// TwinCAT 3 PLC project plc
// Title: ExercicesForPlcProgramming
// Company: Beckhoff Automation Belgium
// ProjectVersion: 1.0.0.0
// Description: Exercices of the book Collection of Exercises for PLC Programming by Tom Mejer Antonson ISBN: 978-87-4305-780-2
// ProgramVersion: 3.1.4026.19
// CompilerDefines: VISU_USEPROPERTYINFO
// libraries:
//   Tc2_ControllerToolbox, * (Beckhoff Automation GmbH)
//   Tc2_Standard, * (Beckhoff Automation GmbH)
//   Tc2_System, * (Beckhoff Automation GmbH)
//   VisuDialogs, * (System)
// project tree:
//   Exercises/02. Logical Circuits/ LogicalCircuits.TcPOU, LogicalCircuits_Ex01.TcPOU, LogicalCircuits_Ex02.TcPOU, LogicalCircuits_Ex03.TcPOU, LogicalCircuits_Ex04.TcPOU, LogicalCircuits_Ex05.TcPOU, LogicalCircuits_Ex06.TcPOU, LogicalCircuits_Ex07.TcPOU, LogicalCircuits_Ex08.TcPOU, LogicalCircuits_Ex09.TcPOU, LogicalCircuits_Ex10.TcPOU, LogicalCircuits_Ex11.TcPOU, LogicalCircuits_Ex12.TcPOU
//   Exercises/03. Safety/ Safety.TcPOU, safety_ex01.TcPOU, safety_ex02.TcPOU
//   Exercises/04. Logic and Counters/ logcacounters_ex2.TcPOU, logcacounters_ex3.TcPOU, logcacounters_ex4.TcPOU, logcacounters_ex5.TcPOU, logcacounters_ex6.TcPOU, logcacounters_ex7.TcPOU, LogicAndCounters.TcPOU, LogicandCountersex01.TcPOU
//   Exercises/05. Timers/ Timers.TcPOU, timers_ex01.TcPOU, timers_ex02.TcPOU, timers_ex03.TcPOU, timers_ex04.TcPOU, timers_ex05.TcPOU, timers_ex06.TcPOU
//   Exercises/06. Analog Signals/ AnalogSignals.TcPOU, analogSignals_ex01.TcPOU, analogSignals_ex02.TcPOU, analogSignals_ex03.TcPOU, analogSignals_ex04.TcPOU, analogSignals_ex05.TcPOU, analogSignals_ex06.TcPOU, analogSignals_ex07.TcPOU, FB_Scale.TcPOU, gemiddelde.TcPOU
//   Exercises/07. Applied Mathematics/ AppliedMathematics.TcPOU, appliedmathematics_ex01.TcPOU
//   Exercises/08. Arrays/ Arrays.TcPOU
//   Exercises/09. Functions and Function Blocks/ FunctionsAndFunctionBlocks.TcPOU, FunctionsAndFunctionBlocksex01.TcPOU, FunctionsAndFunctionBlocksex02.TcPOU, FunctionsAndFunctionBlocksex03.TcPOU
//   Exercises/10. Strings and Structs/ StringsAndStructs.TcPOU
//   Exercises/11. Complex Exercises/ ComplexExercises.TcPOU
//   / GlobalTextList.TcGTLO, MAIN.TcPOU, PlcTask.TcTTO, Visualization Manager.TcVMO (not stored)
//   Project Information/ F_GetCompany.TcPOU, F_GetTitle.TcPOU, F_GetVersion.TcPOU
//   Version/ Global_Version.TcGVL
//   _Library/Inputs/GVLs/ GVL_IO.TcGVL
//   _Library/Inputs/POUs/ DigitalInput_NC.TcPOU, MMotor.TcPOU (not stored), motoroef2_12.TcPOU (not stored), Switch_2P.TcPOU, DigitalInput_NO.TcPOU, DigitalOutput.TcPOU, Switch_4P.TcPOU
//   _Library/Inputs/VISUs/ Visualization.TcVIS
//   _Library/ _TemplateFB.TcPOU
// real-time tasks:
//   TASK PlcTask: cycle T#10ms, priority 20, ADS port 350

CONFIGURATION plc
    RESOURCE PLC ON TwinCAT3
        TASK PlcTask(INTERVAL := T#10ms, PRIORITY := 20);
        PROGRAM MAIN WITH PlcTask : MAIN;
    END_RESOURCE
END_CONFIGURATION

// ---- Version/Global_Version.TcGVL
{attribute 'TcGenerated'}
{attribute 'no-analysis'}
{attribute 'linkalways'}
// This function has been automatically generated from the project information.
VAR_GLOBAL CONSTANT
	{attribute 'const_non_replaced'}
	stLibVersion_ExercicesForPlcProgramming : ST_LibVersion := (iMajor := 1, iMinor := 0, iBuild := 0, iRevision := 0, nFlags := 0, sVersion := '1.0.0.0');
END_VAR

// ---- _Library/Inputs/GVLs/GVL_IO.TcGVL
{attribute 'qualified_only'}
VAR_GLOBAL
	// S1						AT %I*: BOOL;		// S14.2
	// S1						: DigitalInput_NO;   	// S14.2
END_VAR

// ---- MAIN.TcPOU
(*
	Simple solutions for the exercices of the book 
	Collection of Exercises for PLC Programming
	by Tom Mejer Antonson
	ISBN: 978-87-4305-780-2
*)
PROGRAM MAIN
VAR
END_VAR

//LogicalCircuits();
//Safety();
//LogicAndCounters();
//Timers();
AnalogSignals();
//AppliedMathematics();
//Arrays();
//FunctionsAndFunctionBlocks();
//StringsAndStructs();
//ComplexExercises();

END_PROGRAM

// ---- Exercises/06. Analog Signals/AnalogSignals.TcPOU
PROGRAM AnalogSignals

analogSignals_ex07();

END_PROGRAM

// ---- Exercises/06. Analog Signals/analogSignals_ex07.TcPOU
PROGRAM analogSignals_ex07
VAR

	weight				: REAL;
	weightsensor		: REAL;
	hoeveelvaliezen		: INT;
	gemiddeldgewicht	: REAL;
	
	OK					: digitalInput_NO;
	Reset				: digitalInput_NO;
	
	tellersmall			: CTU;
	tellernormal		: CTU;
	tellerbig			: CTU;
	telleroversized		: CTU;
	LIN_TRAFO 			: FB_Scale;
	gemiddelde4			: gemiddelde;
	flankok				: R_trig;
END_VAR

flankok(CLK:= ok.isOn, Q=> );

LIN_TRAFO(
	fIN:= weightsensor, 
	fIN_min:= 4, 
	fIN_max:= 20, 
	fOUT_min:= 0, 
	fOUT_max:= 50, 
	fOUT=> weight);
	
//tellers
	tellersmall(
	CU:= (weight > 0.0) AND (weight <= 5) AND (OK.isOn), 
	RESET:= reset.isOn, 
	PV:= , 
	Q=> , 
	CV=> );
	tellernormal(
	CU:= (weight > 5) AND (weight <= 10) AND (OK.isOn), 
	RESET:= reset.isOn, 
	PV:= , 
	Q=> , 
	CV=> );
	tellerbig(
	CU:= (weight > 10) AND (weight <= 20) AND (OK.isOn), 
	RESET:= reset.isOn, 
	PV:= , 
	Q=> , 
	CV=> );
	telleroversized(
	CU:= (weight > 20) AND (weight <=50) AND (OK.isOn), 
	RESET:= reset.isOn, 
	PV:= , 
	Q=> , 
	CV=> );
	
gemiddelde4(
	fValue:= weight, 
	bAdd:= flankok.Q, 
	bReset:= reset.isOn, 
	fAverage=> gemiddeldgewicht, 
	nCount=> hoeveelvaliezen);

END_PROGRAM

// ---- _Library/Inputs/POUs/DigitalInput_NO.TcPOU
{attribute 'no_explicit_call' := 'do not call this POU directly'} 
FUNCTION_BLOCK DigitalInput_NO
VAR
	DI_Input						AT %I*: BOOL;
END_VAR

PROPERTY isOff : bool
GET
isOff 		:= NOT DI_Input;
END_GET
END_PROPERTY

PROPERTY isOn : bool
GET
isOn			:= DI_Input;
END_GET
END_PROPERTY

END_FUNCTION_BLOCK

// ---- Exercises/06. Analog Signals/FB_Scale.TcPOU
FUNCTION_BLOCK FB_Scale
VAR_INPUT
	fIN				: REAL;
	fIN_min 		: REAL;
	fIN_max			: REAL;
	fOUT_min		: REAL;
	fOUT_max 		: REAL;
END_VAR
VAR_OUTPUT
	fOUT 			: REAL;	
END_VAR
VAR
END_VAR

fOUT := fOUT_min + (fIN - fIN_MIN) * (fOUT_max - fOUT_min) / (fIN_max - fIN_min);

END_FUNCTION_BLOCK

// ---- Exercises/06. Analog Signals/gemiddelde.TcPOU
FUNCTION_BLOCK gemiddelde
VAR_INPUT
	fValue : REAL;                     // Waarde om toe te voegen
    bAdd : BOOL;                       // Trigger om waarde toe te voegen
    bReset : BOOL;                     // Reset de berekening
END_VAR
VAR_OUTPUT
	fAverage : REAL;                   // Gemiddelde waarde
    nCount : INT;                      // Aantal metingen
END_VAR
VAR
	 fSum : REAL := 0.0;                // Som van alle waarden
    bAddOld : BOOL := FALSE;           // Voor edge detectie
	
END_VAR

IF bReset THEN
    nCount := 0;
    fSum := 0.0;
    fAverage := 0.0;
END_IF
IF bAdd AND NOT bAddOld THEN
	fsum := fSum + fValue ;
	nCount := Ncount + 1 ;
	fAverage := fSum / ncount;
END_IF

bAddOld := bAdd;

END_FUNCTION_BLOCK

// ---- Exercises/02. Logical Circuits/LogicalCircuits.TcPOU
PROGRAM LogicalCircuits

//LogicalCircuits_Ex01();
//LogicalCircuits_Ex02();
//LogicalCircuits_Ex03();
//LogicalCircuits_Ex04();
//LogicalCircuits_Ex05();
//LogicalCircuits_Ex06();
//LogicalCircuits_Ex07();
//LogicalCircuits_Ex08();
//LogicalCircuits_Ex09();
LogicalCircuits_Ex10();
//LogicalCircuits_Ex11();
//LogicalCircuits_Ex12();

END_PROGRAM

// ---- Exercises/02. Logical Circuits/LogicalCircuits_Ex10.TcPOU
PROGRAM LogicalCircuits_Ex10
VAR
	S1					: WorkshopLibrary.DigitalInputNO;
	S2					: WorkshopLibrary.DigitalInputNC;
	P1					: WorkshopLibrary.DigitalOutput;
	P2					: WorkshopLibrary.DigitalOutputLatched;
END_VAR

// Evaluate inputs
S1(input := GVL_IO.input01);
S2(input := GVL_IO.input02);

// process outputs
// Solution with standard output
IF S1.isActive	THEN
	P1.on	:= TRUE;
ELSIF S2.isActive	THEN
	P1.on	:= FALSE;
END_IF
P1(output=>GVL_IO.output01);

// Alternative solution with latched output
P2(on:= S1.isActive, off:= S2.isActive, output=> GVL_IO.output02);

END_PROGRAM

// ---- _Library/Inputs/POUs/DigitalOutput.TcPOU
{attribute 'no_explicit_call' := 'do not call this POU directly'} 
FUNCTION_BLOCK DigitalOutput
VAR
	DO_Output					AT %Q*: BOOL;
END_VAR

PROPERTY isOn : bool
GET
isOn				:= DO_Output;
END_GET
END_PROPERTY

METHOD Off : BOOL
DO_Output					:= FALSE;
END_METHOD

METHOD On : BOOL
DO_Output					:= TRUE;
END_METHOD

END_FUNCTION_BLOCK

// ---- Exercises/02. Logical Circuits/LogicalCircuits_Ex01.TcPOU
PROGRAM LogicalCircuits_Ex01
VAR
	S1					: WorkshopLibrary.DigitalInputNO;
	P1					: WorkshopLibrary.DigitalOutput;
END_VAR

// Evaluate inputs
S1(input := GVL_IO.input01);

// process outputs
P1(on:=S1.isActive, output=>GVL_IO.output01);

END_PROGRAM

// ---- Exercises/02. Logical Circuits/LogicalCircuits_Ex02.TcPOU
PROGRAM LogicalCircuits_Ex02
VAR
	S1					: WorkshopLibrary.DigitalInputNO;
	S2					: WorkshopLibrary.DigitalInputNO;
	P1					: WorkshopLibrary.DigitalOutput;
END_VAR

// Evaluate inputs
S1(input := GVL_IO.input01);
S2(input := GVL_IO.input02);

// process outputs
P1(on:=S1.isActive AND S2.isActive, output=>GVL_IO.output01);

END_PROGRAM

// ---- Exercises/02. Logical Circuits/LogicalCircuits_Ex03.TcPOU
PROGRAM LogicalCircuits_Ex03
VAR
	S1					: WorkshopLibrary.DigitalInputNO;
	P1					: WorkshopLibrary.DigitalOutput;
END_VAR

// Evaluate inputs
S1(input := GVL_IO.input01);

// process outputs
IF S1.isActive	THEN
	P1(on:=TRUE, output=>GVL_IO.output01);
END_IF

END_PROGRAM

// ---- Exercises/02. Logical Circuits/LogicalCircuits_Ex04.TcPOU
PROGRAM LogicalCircuits_Ex04
VAR
	S1					: WorkshopLibrary.DigitalInputNO;
	S2					: WorkshopLibrary.DigitalInputNO;
	P1					: WorkshopLibrary.DigitalOutput;
END_VAR

// Evaluate inputs
S1(input := GVL_IO.input01);
S2(input := GVL_IO.input02);

// process outputs
P1(on:=S1.isActive OR S2.isActive, output=>GVL_IO.output01);

END_PROGRAM

// ---- Exercises/02. Logical Circuits/LogicalCircuits_Ex05.TcPOU
PROGRAM LogicalCircuits_Ex05
VAR
	I1					: WorkshopLibrary.DigitalInputNO;
	S1					: WorkshopLibrary.DigitalSwitch;
	P1					: WorkshopLibrary.DigitalOutput;
	P2					: WorkshopLibrary.DigitalOutput;
END_VAR

// Evaluate inputs
I1(input := GVL_IO.input01);
S1(input := I1.isActive);

// process outputs
P1(on:=S1.inPos01, output=>GVL_IO.output01);
P2(on:=S1.inPos01, output=>GVL_IO.output02);

END_PROGRAM

// ---- Exercises/02. Logical Circuits/LogicalCircuits_Ex06.TcPOU
PROGRAM LogicalCircuits_Ex06
VAR
	S1					: WorkshopLibrary.DigitalInputNO;
	P1					: WorkshopLibrary.DigitalOutput;
	P2					: WorkshopLibrary.DigitalOutput;
END_VAR

// Evaluate inputs
S1(input := GVL_IO.input01);

// process outputs
P1(on:=S1.isNotActive, output=>GVL_IO.output01);
P2(on:=S1.isActive, output=>GVL_IO.output02);

END_PROGRAM

// ---- Exercises/02. Logical Circuits/LogicalCircuits_Ex07.TcPOU
PROGRAM LogicalCircuits_Ex07
VAR
	S1					: WorkshopLibrary.DigitalInputNO;
	S2					: WorkshopLibrary.DigitalInputNC;
	P1					: WorkshopLibrary.DigitalOutput;
END_VAR

// Evaluate inputs
S1(input := GVL_IO.input01);
S2(input := GVL_IO.input02);

// process outputs
P1(on:=S1.isActive OR S2.isActive, output=>GVL_IO.output01);

END_PROGRAM

// ---- Exercises/02. Logical Circuits/LogicalCircuits_Ex08.TcPOU
PROGRAM LogicalCircuits_Ex08
VAR
	S1					: WorkshopLibrary.DigitalInputNO;
	S2					: WorkshopLibrary.DigitalInputNO;
	P1					: WorkshopLibrary.DigitalOutput;
	P2					: WorkshopLibrary.DigitalOutput;
	P3					: WorkshopLibrary.DigitalOutput;
END_VAR

// Evaluate inputs
S1(input := GVL_IO.input01);
S2(input := GVL_IO.input02);

// process outputs
P1(on:=S1.isActive AND S2.isNotActive, output=>GVL_IO.output01);
P2(on:=S1.isNotActive AND S2.isActive, output=>GVL_IO.output02);
P3(on:=S1.isActive AND S2.isActive, output=>GVL_IO.output03);

END_PROGRAM

// ---- Exercises/02. Logical Circuits/LogicalCircuits_Ex09.TcPOU
PROGRAM LogicalCircuits_Ex09
VAR
	SX					: WorkshopLibrary.DigitalSwitch4P;
	S1					: WorkshopLibrary.DigitalInputNO;
	S2					: WorkshopLibrary.DigitalInputNO;
	S3					: WorkshopLibrary.DigitalInputNO;
	P1					: WorkshopLibrary.DigitalOutput;
	P2					: WorkshopLibrary.DigitalOutput;
	P3					: WorkshopLibrary.DigitalOutput;
END_VAR

// Evaluate inputs
S1(input := GVL_IO.input01);
S2(input := GVL_IO.input02);
S3(input := GVL_IO.input03);
SX(
	input01	:= S1.isActive, 
	input02	:= S2.isActive, 
	input03	:= S3.isActive, 
	inPos00	=> , 
	inPos01	=> , 
	inPos02	=> , 
	inPos03	=> );

// process outputs
P1(on:=SX.inPos01 OR SX.inPos03, output=>GVL_IO.output01);
P2(on:=SX.inPos02 OR SX.inPos03, output=>GVL_IO.output02);
P3(on:=SX.inPos03, output=>GVL_IO.output03);

END_PROGRAM

// ---- Exercises/02. Logical Circuits/LogicalCircuits_Ex11.TcPOU
PROGRAM LogicalCircuits_Ex11
VAR
	S1stand 				: Switch_2P;
	sensor			 		: digitalInput_NO;
	
	motor: MMotor;
END_VAR



motor(start:=(S1stand.position0 and sensor.isOff) , stop:= (S1stand.position1 or sensor.isOn), motor=> );

END_PROGRAM

// ---- _Library/Inputs/POUs/Switch_2P.TcPOU
FUNCTION_BLOCK Switch_2P
VAR_INPUT
END_VAR
VAR_OUTPUT
END_VAR
VAR
	DI_Input at %I* : bool;
END_VAR

PROPERTY position0 : BOOL
GET
position0 := not DI_Input;
END_GET
END_PROPERTY

PROPERTY position1 : BOOL
GET
position1 := DI_Input;
END_GET
END_PROPERTY

END_FUNCTION_BLOCK

// ---- Exercises/02. Logical Circuits/LogicalCircuits_Ex12.TcPOU
PROGRAM LogicalCircuits_Ex12
VAR
	sensorB2		 		: digitalInput_NO;
	sensorB1		 		: digitalInput_NO;
	S1				 		: digitalInput_NO;
	S2				 		: digitalInput_NO;
	
	
END_VAR

END_PROGRAM

// ---- Exercises/03. Safety/Safety.TcPOU
PROGRAM Safety

END_PROGRAM

// ---- Exercises/03. Safety/safety_ex01.TcPOU
PROGRAM safety_ex01
VAR
	
B1				: digitalInput_NO; 
B2				: digitalInput_NO; 
B3				: digitalInput_NO; 
B4				: digitalInput_NO; 

Q4				: DigitalOutput := TRUE;

RFB2			: R_trig;
FFB4			: F_trig;


END_VAR

RFB2(clk := B2);
FFB4(clk := B4);

//afgaan bij het toekomen van de palet 
IF B1.isOn AND RFB2.Q THEN
	Q4.Off();
END_IF

IF NOT B3 AND FFB4.Q THEN
	Q4.On();
END_IF

END_PROGRAM

// ---- Exercises/03. Safety/safety_ex02.TcPOU
PROGRAM safety_ex02
VAR

M1 					: DigitalOutput;
M1_start			: digitalInput_NO;
M1_stop				: digitalInput_NC;
M1_stop_safe		: digitalInput_NC;
M2					: digitalOutput; 
M4					: digitaloutput;
M5					: digitaloutput;
S1					: digitalInput_NO; 
S2					: digitalInput_NC;
S3					: digitalInput_NO; 
S6					: digitalInput_NC;
S7					: digitalInput_NC;
B4					: digitalInput_NO;
B5					: digitalInput_NO;
P1					: digitaloutput;
P2					: digitaloutput;
P3					: digitaloutput;
P4					: digitaloutput;

END_VAR

//noodstoppen
IF S2.broken OR S6.broken OR S7.broken OR M1_STOP_SAFE.broken OR M1_stop.broken OR S1.isOff THEN
	M1.Off();
END_IF
IF S6.broken OR S7.broken THEN
	P4.On();
END_IF

//noodstop resetten
IF S6.broken OR S7.broken THEN
	P4.On();
END_IF
IF S3.isOn THEN
	P4.Off();
END_IF


//start					//alle stoppen												//veiligheidsdeuren				//start drukknoppen
IF (S2.in_dienst AND M1_STOP_SAFE.in_dienst AND M1_STOP.in_dienst AND P4.Off) AND (B4.isOn AND B5.isOn) AND M1_start.isOn OR S1.isOn THEN
	M1.On();
	M2.On();
END_IF


//stop van de band 
IF S2.broken OR P4.On THEN
	M2.Off();
	P1.On();
END_IF



//veiligheidsdeuren
if S2.broken OR S6.broken OR S7.broken THEN
	M4.On();	(*on betekent dat ze open kunnen*)
	M5.On();	(*on betekent dat ze open kunnen*)
ELSE 
	M4.Off();	(*off betekent dat ze niet open kunnen*)
	M5.Off();	(*off betekent dat ze niet open kunnen*)
END_IF

//sensoren die checken of de deuren toe zijn

IF B4.isOff (*off betekent dat hij geen signaal krijgt dus deur is open*) OR B5.isOff THEN
	P1.On();
ELSE 
	P1.Off();
END_IF

// lamp robot actief
IF M1.On THEN
	P2.On();
ELSE 
	P2.Off();
END_IF

IF S2.broken THEN
	P3.On();
END_IF
IF S1.isOn THEN
	P3.Off();
END_IF

END_PROGRAM

// ---- _Library/Inputs/POUs/DigitalInput_NC.TcPOU
FUNCTION_BLOCK DigitalInput_NC
VAR_INPUT
END_VAR
VAR_OUTPUT
END_VAR
VAR
	DIinputNC at %I* : bool;
END_VAR

PROPERTY broken : BOOL
GET
broken := DIinputNC;
END_GET
END_PROPERTY

PROPERTY in_dienst : BOOL
GET
in_dienst := not DIinputNC;
END_GET
END_PROPERTY

END_FUNCTION_BLOCK

// ---- Exercises/04. Logic and Counters/logcacounters_ex2.TcPOU
PROGRAM logcacounters_ex2
VAR
	S1				: DigitalInput_NO;
	S2				: DigitalInput_NO;
	P1				: DigitalOutput;
	CV 				: INT := 0;
	S1flank 		: R_trig;
END_VAR

S1flank(clk := S1.isOn);

IF S1flank.Q THEN
	CV := CV + 1; 
END_IF 
IF CV >= 4 THEN
	P1.On();
END_IF
IF S2.isOn THEN
	CV := 0;
	P1.Off();
END_IF

END_PROGRAM

// ---- Exercises/04. Logic and Counters/logcacounters_ex3.TcPOU
PROGRAM logcacounters_ex3
VAR
	S1				: DigitalInput_NO;
	P1				: DigitalOutput;
	CV 				: INT := 0;
	S1flank 		: R_trig;
END_VAR

S1flank(clk := S1.isOn);

IF S1flank.Q THEN
	CV := CV + 1; 
END_IF 
IF CV >= 5 THEN
	P1.On();
END_IF
IF CV = 10 THEN
	CV := 0;
	P1.Off();
END_IF

END_PROGRAM

// ---- Exercises/04. Logic and Counters/logcacounters_ex4.TcPOU
PROGRAM logcacounters_ex4
VAR
	S1				: DigitalInput_NO;
	CV 				: INT := 0;
	
	P1 				: DigitalOutput;
	P2 				: DigitalOutput;
	P3 				: DigitalOutput;
	P4 				: DigitalOutput;
	
	S1flank 		: R_trig;
END_VAR

S1flank(clk := S1.isOn);

IF S1flank.Q THEN
	CV := CV + 1;
END_IF

IF CV = 1 THEN P1.On(); END_IF
IF CV = 2 THEN P1.On(); P2.On(); END_IF
IF CV = 3 THEN P1.On(); P2.On(); P3.On(); END_IF
IF CV = 4 THEN P1.On(); P2.On(); P3.On(); P4.On() ; END_IF
IF CV = 0 THEN P1.off(); P2.off(); P3.off(); P4.off() ; END_IF

IF CV > 4 THEN
	CV := 0;
END_IF

END_PROGRAM

// ---- Exercises/04. Logic and Counters/logcacounters_ex5.TcPOU
PROGRAM logcacounters_ex5
VAR
	
S1				: DigitalInput_NO;
S2				: DigitalInput_NO;
P1 				: DigitalOutput;
CV1 				: INT := 0;
CV2 				: INT := 0;
S1flank 		: R_trig;
S2flank 		: R_trig;
END_VAR

S1flank(clk := S1.isOn);
S2flank(clk := S2.isOn);


IF S1flank.Q THEN
	cv1 := cv1 + 1;
END_IF
IF S2flank.Q THEN
	CV2 := CV2 + 1;
END_IF
IF CV1 = 4 AND CV2 = 5 THEN
	P1.On();
END_IF
IF S1.isOn AND S2.isOn THEN 
	CV1 := 0;
	CV2 := 0;
END_IF

END_PROGRAM

// ---- Exercises/04. Logic and Counters/logcacounters_ex6.TcPOU
PROGRAM logcacounters_ex6
VAR
	S1				: DigitalInput_NO;
	S2				: DigitalInput_NO;
	P1 				: DigitalOutput;
	CV1 				: INT := 0;
	CV2 				: INT := 0;
	S1flank 		: R_trig;
	S2flank 		: R_trig;
END_VAR

S1flank(clk := S1.isOn);
S2flank(clk := S2.isOn);


IF S1flank.Q THEN
	cv1 := cv1 + 1;
END_IF
IF S2flank.Q THEN
	CV2 := CV2 + 1;
END_IF
IF CV1 = 4 AND CV2 = 5 THEN
	P1.On();
END_IF
IF S1.isOn AND S2.isOn THEN 
	CV1 := 0;
	CV2 := 0;
END_IF

//vervolg voor de volgende oefening 
IF CV1 > 6 THEN
	P1.Off(); CV1 := 0;
END_IF
IF CV2 > 6 THEN
	P1.Off(); CV2 := 0;
END_IF

END_PROGRAM

// ---- Exercises/04. Logic and Counters/logcacounters_ex7.TcPOU
PROGRAM logcacounters_ex7
VAR
	B11				: DigitalInput_NO;
	B2				: DigitalInput_NO;
	B3				: DigitalInput_NO;
	
	M1				: digitaloutput;
	p1				: digitaloutput;
	P2				: digitaloutput;
	
	teller			: CTUD;
	B1F				: R_trig;
	B2F				: R_trig;
	B3F				: R_trig;
	B2FF			: F_trig;
	
END_VAR

B1F(clk := B11);
B2F(clk := B2);
B3F(clk := B3);
B2FF(clk := B2);


	
//openen en sluiten slagboom
IF B11.isOn THEN
	M1.On();
END_IF
IF B2FF.Q THEN
	M1.Off();
END_IF

END_PROGRAM

// ---- Exercises/04. Logic and Counters/LogicAndCounters.TcPOU
PROGRAM LogicAndCounters

END_PROGRAM

// ---- Exercises/04. Logic and Counters/LogicandCountersex01.TcPOU
PROGRAM LogicandCountersex01
VAR
	S1				: DigitalInput_NO;
	P1				: DigitalOutput;
	CV				: INT  := 0;
	S1_flank		: R_trig;
END_VAR

S1_flank(clk := S1.isOn);

IF S1_flank.Q THEN
	CV := CV + 1;
END_IF

IF CV >= 5 THEN
	P1.On();
END_IF

END_PROGRAM

// ---- Exercises/05. Timers/Timers.TcPOU
PROGRAM Timers

END_PROGRAM

// ---- Exercises/05. Timers/timers_ex01.TcPOU
FUNCTION_BLOCK timers_ex01
VAR_INPUT
	stand			: Switch_2P;
END_VAR
VAR_OUTPUT
	P1				: DigitalOutput;
END_VAR
VAR
	Timer1			: TON;
END_VAR

Timer1(IN:= stand.position1, PT:= T#5S, Q=> , ET=> );

IF Timer1.Q THEN
	P1.On();
END_IF

END_FUNCTION_BLOCK

// ---- Exercises/05. Timers/timers_ex02.TcPOU
FUNCTION_BLOCK timers_ex02
VAR_INPUT
	S1				: DigitalInput_NO;
END_VAR
VAR_OUTPUT
	P1				: DigitalOutput;
END_VAR
VAR
	Timer1_ex02		: TOF;
END_VAR

Timer1_ex02(IN:= S1.isOn, PT:= T#10S, Q=> , ET=> );

IF S1.isOn THEN
	P1.On();
END_IF
IF Timer1_ex02.Q THEN
	P1.Off();
END_IF

END_FUNCTION_BLOCK

// ---- Exercises/05. Timers/timers_ex03.TcPOU
FUNCTION_BLOCK timers_ex03
VAR_INPUT
	stand			: Switch_2P;
END_VAR
VAR_OUTPUT
	P1				: DigitalOutput;
END_VAR
VAR
	Timer1_ex03		: TOF;
	Timer2_ex03		: TON;
END_VAR

END_FUNCTION_BLOCK

// ---- Exercises/05. Timers/timers_ex04.TcPOU
FUNCTION_BLOCK timers_ex04
VAR_INPUT
	stand			: Switch_2P;
END_VAR
VAR_OUTPUT
	P1				: DigitalOutput;
	P2				: DigitalOutput;
END_VAR
VAR
	Timer1_ex04		: TON;
	Timer2_ex04		: Tof; 
END_VAR

Timer1_ex04(IN:= stand.position1, PT:= T#10S, Q=> , ET=> );
Timer2_ex04(IN:= P2.On, PT:= T#10S , Q=> , ET=> );
IF stand.position1 THEN
	P1.On();
END_IF
IF Timer1_ex04.Q THEN
	P1.On();
	P2.On();
END_IF
IF Timer2_ex04.Q THEN
	P1.Off();
	P2.Off();
END_IF

END_FUNCTION_BLOCK

// ---- Exercises/05. Timers/timers_ex05.TcPOU
FUNCTION_BLOCK timers_ex05
VAR_INPUT
	stand			: Switch_2P;
END_VAR
VAR_OUTPUT
	P1				: DigitalOutput;
	P2				: DigitalOutput;
END_VAR
VAR
	Timer1_ex04		: TON;
	Timer2_ex04		: Tof; 
END_VAR

END_FUNCTION_BLOCK

// ---- Exercises/05. Timers/timers_ex06.TcPOU
FUNCTION_BLOCK timers_ex06
VAR_INPUT
	stand			: Switch_2P;
END_VAR
VAR_OUTPUT
	P1				: DigitalOutput;
	P2				: DigitalOutput;
END_VAR
VAR
	Timer1_ex04		: TON;
	Timer2_ex04		: Tof; 
END_VAR

END_FUNCTION_BLOCK

// ---- Exercises/06. Analog Signals/analogSignals_ex01.TcPOU
PROGRAM analogSignals_ex01
VAR
	Frawsensor		: REAL;
	fScaledvalue	: real;
	
	LIN_TRAFO 		: FB_Scale;
END_VAR

LIN_TRAFO(
	fIN:= frawsensor, 
	fIN_min:= 4, 
	fIN_max:= 20, 
	fOUT_min:= 0, 
	fOUT_max:= 100, 
	fOUT=> fScaledvalue);

END_PROGRAM

// ---- Exercises/06. Analog Signals/analogSignals_ex02.TcPOU
PROGRAM analogSignals_ex01_1
VAR
	Frawsensor		: REAL;
	fScaledvalue	: real;
	
	LIN_TRAFO 		: FB_Scale;
END_VAR

LIN_TRAFO(
	fIN:= frawsensor, 
	fIN_min:= 4, 
	fIN_max:= 20, 
	fOUT_min:= 0, 
	fOUT_max:= 100, 
	fOUT=> fScaledvalue);

END_PROGRAM

// ---- Exercises/06. Analog Signals/analogSignals_ex03.TcPOU
PROGRAM analogSignals_ex02_1
VAR
	Frawsensor			: REAL;
	potentiometervalue	: REAL;
	
	LIN_TRAFO 			: FB_Scale;
END_VAR

LIN_TRAFO(
	fIN:= frawsensor, 
	fIN_min:= 0, 
	fIN_max:= 20, 
	fOUT_min:= 0, 
	fOUT_max:= 60, 
	fOUT=> potentiometervalue);

END_PROGRAM

// ---- Exercises/06. Analog Signals/analogSignals_ex04.TcPOU
PROGRAM analogSignals_ex03_1
VAR
	Frawsensor			: REAL;
	weight				: REAL;
	
	LIN_TRAFO 			: FB_Scale;
END_VAR

LIN_TRAFO(
	fIN:= frawsensor, 
	fIN_min:= 0, 
	fIN_max:= 10, 
	fOUT_min:= 0, 
	fOUT_max:= 500, 
	fOUT=> weight);

END_PROGRAM

// ---- Exercises/06. Analog Signals/analogSignals_ex05.TcPOU
PROGRAM analogSignals_ex05
VAR
	rpmcontrol			: REAL;
	rpm					: REAL;
	
	LIN_TRAFO 			: FB_Scale;
END_VAR

LIN_TRAFO(
	fIN:= rpmcontrol, 
	fIN_min:= 0, 
	fIN_max:= 120, 
	fOUT_min:= 4, 
	fOUT_max:= 20, 
	fOUT=> rpm);

END_PROGRAM

// ---- Exercises/06. Analog Signals/analogSignals_ex06.TcPOU
PROGRAM analogSignals_ex06
VAR
	valvecontrol			: REAL;
	valveopening			: REAL;
	
	LIN_TRAFO 			: FB_Scale;
END_VAR

LIN_TRAFO(
	fIN:= valvecontrol, 
	fIN_min:= 0, 
	fIN_max:= 100, 
	fOUT_min:= 0, 
	fOUT_max:= 10, 
	fOUT=> valveopening);

END_PROGRAM

// ---- Exercises/07. Applied Mathematics/AppliedMathematics.TcPOU
PROGRAM AppliedMathematics

END_PROGRAM

// ---- Exercises/07. Applied Mathematics/appliedmathematics_ex01.TcPOU
PROGRAM appliedmathematics_ex01
VAR
// Cylinder dimensions
    cHeight : LREAL := 2.75;        // Height/Length of cylinder in meters
    cDiameter : LREAL := 1.4;       // Diameter of cylinder in meters
    cRadius : LREAL;                // Calculated radius
    
    // Sensor input
    fSensorRaw : LREAL;             // Raw sensor value (e.g., 4-20mA, 0-10V)
    fbLevelTrafo : FB_lin_trafo;    // Linear transformation instance
    
    // Calculated values
    fLiquidHeight : LREAL;          // Current liquid level in meters
    fVolumeLiters : LREAL;          // Volume in liters
    fVolumeCubicMeters : LREAL;     // Volume in m³
    fFillPercentage : LREAL;        // Fill percentage
    fMaxVolume : LREAL;             // Maximum cylinder volume
    
    // Configuration
    bVerticalCylinder : BOOL := TRUE;   // TRUE = vertical, FALSE = horizontal
    fSensorMin : LREAL := 4.0;          // Sensor minimum (e.g., 4mA)
    fSensorMax : LREAL := 20.0;         // Sensor maximum (e.g., 20mA)
END_VAR

END_PROGRAM

// ---- Exercises/08. Arrays/Arrays.TcPOU
PROGRAM Arrays

END_PROGRAM

// ---- Exercises/09. Functions and Function Blocks/FunctionsAndFunctionBlocks.TcPOU
PROGRAM FunctionsAndFunctionBlocks

END_PROGRAM

// ---- Exercises/09. Functions and Function Blocks/FunctionsAndFunctionBlocksex01.TcPOU
PROGRAM FunctionsAndFunctionBlocksex01
VAR
number1 		: number;
number2			: number;
sum12			: number;
END_VAR

number1 + number2 := sum12;

END_PROGRAM

// ---- Exercises/09. Functions and Function Blocks/FunctionsAndFunctionBlocksex02.TcPOU
PROGRAM FunctionsAndFunctionBlocksex02
VAR
number1 		: number;
number2			: number;
sum12			: number;
END_VAR

number1 * number2 := sum12;

END_PROGRAM

// ---- Exercises/09. Functions and Function Blocks/FunctionsAndFunctionBlocksex03.TcPOU
FUNCTION_BLOCK FunctionsAndFunctionBlocksex03
VAR_INPUT
	number1 		: number;
	number2 		: number;
END_VAR
VAR_OUTPUT
	sum12 			: number;
	counter 		: number;
END_VAR
VAR
END_VAR

END_FUNCTION_BLOCK

// ---- Exercises/10. Strings and Structs/StringsAndStructs.TcPOU
PROGRAM StringsAndStructs

END_PROGRAM

// ---- Exercises/11. Complex Exercises/ComplexExercises.TcPOU
PROGRAM ComplexExercises

END_PROGRAM

// ---- Project Information/F_GetCompany.TcPOU
// This function has been automatically generated from the project information.
{attribute 'signature_flag' := '1073741824'}
{attribute 'TcGenerated'}
{attribute 'no-analysis'}
FUNCTION F_GetCompany : WSTRING
VAR_INPUT
	
END_VAR

F_GetCompany := "Beckhoff Automation Belgium";

END_FUNCTION

// ---- Project Information/F_GetTitle.TcPOU
// This function has been automatically generated from the project information.
{attribute 'signature_flag' := '1073741824'}
{attribute 'TcGenerated'}
{attribute 'no-analysis'}
FUNCTION F_GetTitle : WSTRING
VAR_INPUT
	
END_VAR

F_GetTitle := "ExercicesForPlcProgramming";

END_FUNCTION

// ---- Project Information/F_GetVersion.TcPOU
// This function has been automatically generated from the project information.
{attribute 'signature_flag' := '1073741824'}
{attribute 'TcGenerated'}
{attribute 'no-analysis'}
FUNCTION F_GetVersion : ST_LibVersion
VAR_INPUT
	
END_VAR

F_GetVersion.iMajor := 1;
F_GetVersion.iMinor := 0;
F_GetVersion.iBuild := 0;
F_GetVersion.iRevision := 0;
F_GetVersion.sVersion := '1.0.0.0';
F_GetVersion.nFlags := 0;

END_FUNCTION

// ---- _Library/Inputs/POUs/Switch_4P.TcPOU
FUNCTION_BLOCK Switch_4P
VAR_INPUT
END_VAR
VAR_OUTPUT
END_VAR
VAR
	DIinput AT %I* : BOOL;
	DIinput2 AT %I* : BOOL;
	DIinput3 at %I* : bool;
END_VAR

PROPERTY Po0 : BOOL
GET
Po0 := not DIinput;
END_GET
END_PROPERTY

PROPERTY Po1 : BOOL
GET
Po1 := DIinput;
END_GET
END_PROPERTY

PROPERTY Po2 : BOOL
GET
Po2 := DIinput2;
END_GET
END_PROPERTY

PROPERTY Po3 : BOOL
GET
Po3 := DIinput3;
END_GET
END_PROPERTY

END_FUNCTION_BLOCK

// ---- _Library/_TemplateFB.TcPOU
{attribute 'no_explicit_call' := 'do not call this POU directly, call execute'} 
FUNCTION_BLOCK _TemplateFB
VAR
END_VAR

// NO CODE HERE, USE execute

METHOD execute
END_METHOD

END_FUNCTION_BLOCK

// ---- GlobalTextList.TcGTLO
TEXTLIST GlobalTextList
  538 = '%5.2f'
  227 = 'big: %d'
  931 = 'gemiddelde: %5.2f'
  154 = 'hoeveel valiezen: %d'
  933 = 'normal: %d'
  928 = 'oversized: %d'
  46 = 'small: %d'
  415 = 'valies: %5.2f'
END_TEXTLIST

// ---- _Library/Inputs/VISUs/Visualization.TcVIS
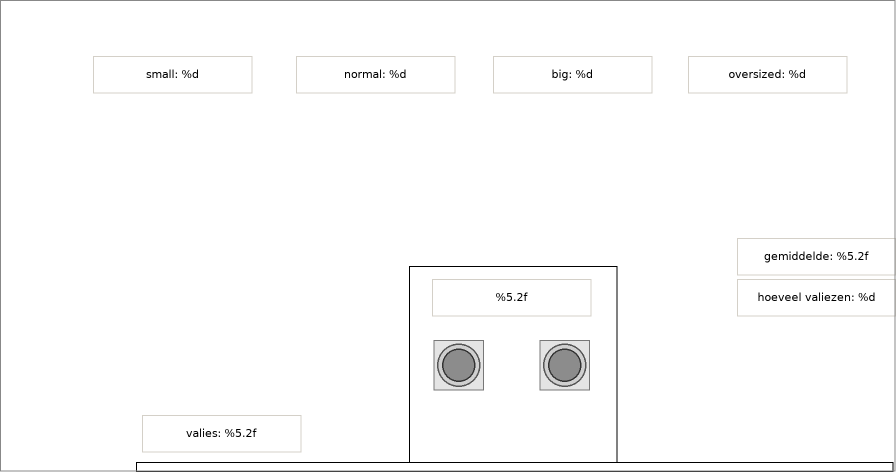
VISUALIZATION Visualization  // 896x472
    Rectangle (409,266 208x206)
    PushSwitch (432,340 53x50), variable: analogSignals_ex07.OK.DI_Input, behaviour: TOGGLE, style: Switch-PushSwitch-Gray
    PushSwitch (538,340 53x50), variable: analogSignals_ex07.Reset.DI_Input, behaviour: TOGGLE, style: Switch-PushSwitch-Gray
    Rectangle (136,462 757x10)
    Textfield (432,279 159x37), "%5.2f", text variable: analogSignals_ex07.weight
    Textfield (93,56 159x37), "small: %d", text variable: analogSignals_ex07.tellersmall.CV
    Textfield (296,56 159x37), "normal: %d", text variable: analogSignals_ex07.tellernormal.CV
    Textfield (493,56 159x37), "big: %d", text variable: analogSignals_ex07.tellerbig.CV
    Textfield (688,56 159x37), "oversized: %d", text variable: analogSignals_ex07.telleroversized.CV
    Textfield (737,238 159x37), "gemiddelde: %5.2f", text variable: analogSignals_ex07.gemiddelde4.fAverage
    Textfield (737,279 159x37), "hoeveel valiezen: %d", text variable: analogSignals_ex07.gemiddelde4.nCount
    Textfield (142,415 159x37), "valies: %5.2f", text variable: analogSignals_ex07.weightsensor
        OnMouseClick: write the text variable via VisuDialogs.Numpad, min 4, max 20
END_VISUALIZATION
